PROGRAM Main
VAR
END_VAR

END_PROGRAM

(* stored: Version 1.1.0.1, ProductVersion 3.1.4024.0
   POU Main: Id {7de81d17-9477-439d-b1f6-5157a4a2df6c}, SpecialFunc None *)
